Fanuc TP program (LS listing): calib_sph.ls

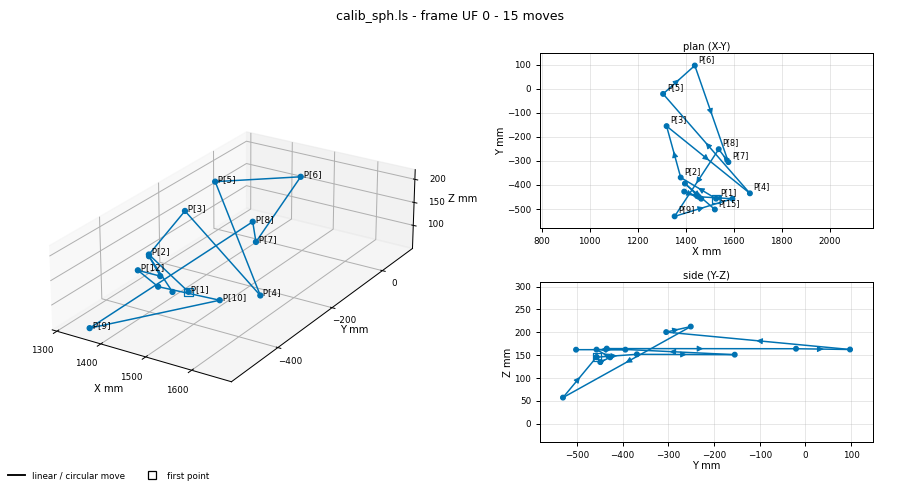
[picture p0: tool path of calib_sph.ls in frame UF 0, 15 of 15 moves have a stored position in this frame; points joined in program order, loops and branches not executed]
/PROG  CALIB_SPH
/ATTR
OWNER		= MNEDITOR;
COMMENT		= "";
PROG_SIZE	= 1683;
CREATE		= DATE 25-09-23  TIME 10:26:52;
MODIFIED	= DATE 25-09-23  TIME 12:20:10;
FILE_NAME	= ;
VERSION		= 0;
LINE_COUNT	= 38;
MEMORY_SIZE	= 2039;
PROTECT		= READ_WRITE;
TCD:  STACK_SIZE	= 0,
      TASK_PRIORITY	= 50,
      TIME_SLICE	= 0,
      BUSY_LAMP_OFF	= 0,
      ABORT_REQUEST	= 0,
      PAUSE_REQUEST	= 0;
DEFAULT_GROUP	= 1,*,*,*,*;
CONTROL_CODE	= 00000000 00000000;
/APPL
/MN
   1:  UTOOL_NUM=10 ;
   2:  UFRAME_NUM=0 ;
   3:  OVERRIDE=30% ;
   4:   ;
   5:L P[1] 300mm/sec FINE    ;
   6:  CALL GRAB_CAL    ;
   7:L P[2] 300mm/sec FINE    ;
   8:  CALL GRAB_CAL    ;
   9:L P[3] 300mm/sec FINE    ;
  10:  CALL GRAB_CAL    ;
  11:   ;
  12:L P[4] 300mm/sec FINE    ;
  13:  CALL GRAB_CAL    ;
  14:L P[5] 300mm/sec FINE    ;
  15:  CALL GRAB_CAL    ;
  16:L P[6] 300mm/sec FINE    ;
  17:  CALL GRAB_CAL    ;
  18:   ;
  19:L P[7] 300mm/sec FINE    ;
  20:  CALL GRAB_CAL    ;
  21:L P[8] 300mm/sec FINE    ;
  22:  CALL GRAB_CAL    ;
  23:L P[9] 300mm/sec FINE    ;
  24:  CALL GRAB_CAL    ;
  25:   ;
  26:L P[10] 300mm/sec FINE    ;
  27:  CALL GRAB_CAL    ;
  28:L P[11] 300mm/sec FINE    ;
  29:  CALL GRAB_CAL    ;
  30:L P[12] 300mm/sec FINE    ;
  31:  CALL GRAB_CAL    ;
  32:   ;
  33:L P[13] 300mm/sec FINE    ;
  34:  CALL GRAB_CAL    ;
  35:L P[14] 300mm/sec FINE    ;
  36:  CALL GRAB_CAL    ;
  37:L P[15] 300mm/sec FINE    ;
  38:  CALL GRAB_CAL    ;
/POS
P[1]{
   GP1:
	UF : 0, UT : 10,		CONFIG : 'F U T, 0, 0, -1',
	X =  1526.735  mm,	Y =  -457.029  mm,	Z =   145.665  mm,
	W =  -122.482 deg,	P =    87.522 deg,	R =   -34.898 deg
};
P[2]{
   GP1:
	UF : 0, UT : 10,		CONFIG : 'F U T, 0, 0, -1',
	X =  1379.474  mm,	Y =  -368.840  mm,	Z =   151.932  mm,
	W =  -122.809 deg,	P =    87.518 deg,	R =   -73.811 deg
};
P[3]{
   GP1:
	UF : 0, UT : 10,		CONFIG : 'F U T, 0, 0, -1',
	X =  1320.693  mm,	Y =  -154.795  mm,	Z =   151.145  mm,
	W =  -123.900 deg,	P =    87.487 deg,	R =  -114.175 deg
};
P[4]{
   GP1:
	UF : 0, UT : 10,		CONFIG : 'F U T, 0, 0, -1',
	X =  1667.578  mm,	Y =  -434.741  mm,	Z =   164.454  mm,
	W =  -122.472 deg,	P =    87.525 deg,	R =   -16.614 deg
};
P[5]{
   GP1:
	UF : 0, UT : 10,		CONFIG : 'F U T, 0, 0, 0',
	X =  1306.189  mm,	Y =   -20.676  mm,	Z =   164.136  mm,
	W =  -122.929 deg,	P =    87.509 deg,	R =  -136.322 deg
};
P[6]{
   GP1:
	UF : 0, UT : 10,		CONFIG : 'F U T, 0, 0, 0',
	X =  1438.150  mm,	Y =    97.502  mm,	Z =   162.464  mm,
	W =  -122.629 deg,	P =    87.516 deg,	R =  -168.964 deg
};
P[7]{
   GP1:
	UF : 0, UT : 10,		CONFIG : 'F U T, 0, 0, -1',
	X =  1578.127  mm,	Y =  -304.732  mm,	Z =   200.524  mm,
	W =  -171.512 deg,	P =    72.136 deg,	R =   -83.323 deg
};
P[8]{
   GP1:
	UF : 0, UT : 10,		CONFIG : 'F U T, 0, 0, -1',
	X =  1537.801  mm,	Y =  -250.965  mm,	Z =   212.664  mm,
	W =  -173.404 deg,	P =    65.461 deg,	R =   -85.090 deg
};
P[9]{
   GP1:
	UF : 0, UT : 10,		CONFIG : 'F U T, 0, 0, -1',
	X =  1354.139  mm,	Y =  -530.601  mm,	Z =    57.247  mm,
	W =    -4.246 deg,	P =    72.542 deg,	R =    63.482 deg
};
P[10]{
   GP1:
	UF : 0, UT : 10,		CONFIG : 'F U T, 0, 0, -1',
	X =  1594.819  mm,	Y =  -457.137  mm,	Z =   145.731  mm,
	W =    99.231 deg,	P =    78.842 deg,	R =  -172.715 deg
};
P[11]{
   GP1:
	UF : 0, UT : 10,		CONFIG : 'F U T, 0, 0, -1',
	X =  1454.151  mm,	Y =  -448.977  mm,	Z =   134.898  mm,
	W =   -93.848 deg,	P =    76.628 deg,	R =    -6.140 deg
};
P[12]{
   GP1:
	UF : 0, UT : 10,		CONFIG : 'F U T, 0, 0, -1',
	X =  1394.159  mm,	Y =  -427.426  mm,	Z =   145.320  mm,
	W =   -93.884 deg,	P =    76.651 deg,	R =   -23.636 deg
};
P[13]{
   GP1:
	UF : 0, UT : 10,		CONFIG : 'F U T, 0, 0, -1',
	X =  1464.866  mm,	Y =  -457.133  mm,	Z =   162.239  mm,
	W =  -122.345 deg,	P =    87.512 deg,	R =   -34.452 deg
};
P[14]{
   GP1:
	UF : 0, UT : 10,		CONFIG : 'F U T, 0, 0, -1',
	X =  1397.071  mm,	Y =  -394.007  mm,	Z =   162.150  mm,
	W =  -122.426 deg,	P =    87.516 deg,	R =   -34.533 deg
};
P[15]{
   GP1:
	UF : 0, UT : 10,		CONFIG : 'F U T, 0, 0, -1',
	X =  1521.744  mm,	Y =  -501.955  mm,	Z =   162.046  mm,
	W =  -122.498 deg,	P =    87.522 deg,	R =   -34.606 deg
};
/END
